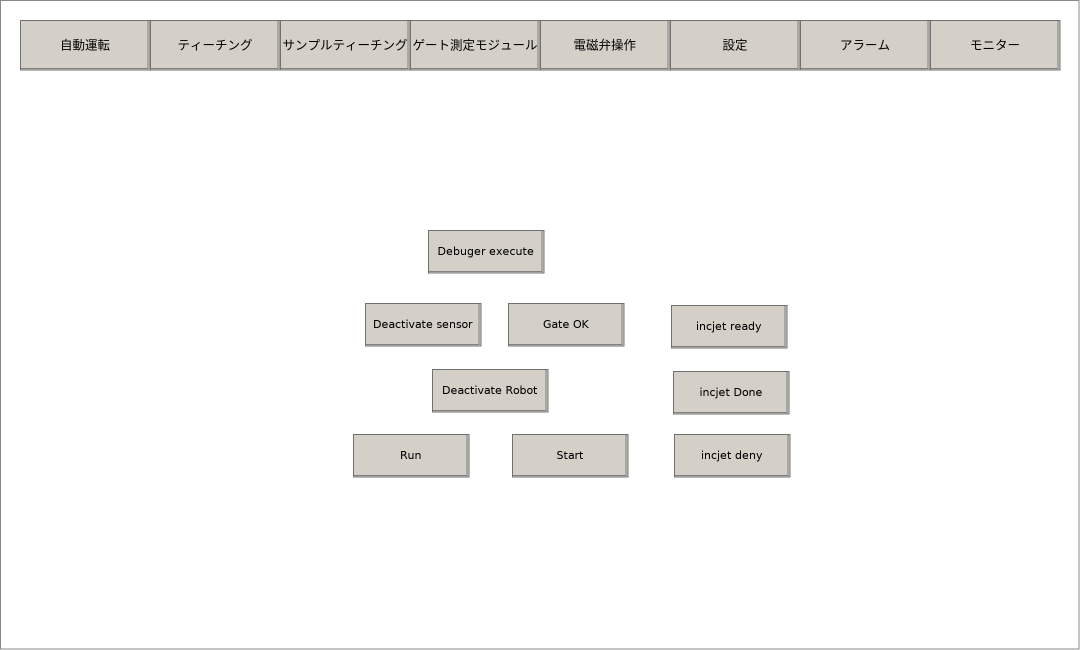
VISUALIZATION s_debug  // 1080x650
    Rectangle (0,0 1080x650)
    Button (20,20 130x50), "自動運転"
        OnMouseClick: change screen: s_auto
    Button (150,20 130x50), "ティーチング"
        OnMouseClick: change screen: s_teaching1
    Button (670,20 130x50), "設定"
        OnMouseClick: change screen: s_setting
    Button (540,20 130x50), "電磁弁操作"
        OnMouseClick: change screen: s_manual
    Button (410,20 130x50), "ゲート測定モジュール"
        OnMouseClick: change screen: s_gm_teaching
    Button (800,20 130x50), "アラーム", colour toggle: gvl_io.flg_signalTowerRed
        OnMouseClick: change screen: s_alarm
    Button (280,20 130x50), "サンプルティーチング"
        OnMouseClick: change screen: s_sample
    Button (930,20 130x50), "モニター"
        OnMouseClick: change screen: s_monitor
    Button (365,303 116x43), "Deactivate sensor", colour toggle: gvl_visu.flg_btn_vacSensOn
        toggle gvl_visu.flg_btn_vacSensOn
    Button (428,230 116x43), "Debuger execute", colour toggle: gvl_debug.flg_debug_run
        toggle gvl_debug.flg_debug_run
    Button (353,434 116x43), "Run", colour toggle: gvl_debug.flg_debug_start
        toggle gvl_debug.flg_debug_start
    Button (508,303 116x43), "Gate OK", colour toggle: gvl_debug.gateLengthISSuccessed
        toggle gvl_debug.gateLengthISSuccessed
    Button (512,434 116x43), "Start", colour toggle: gvl_debug.lensSetDone
        toggle gvl_debug.lensSetDone
    Button (671,305 116x43), "incjet ready", colour toggle: gvl_debug.flg_stampReady
        toggle gvl_debug.flg_stampReady
    Button (673,371 116x43), "incjet Done", colour toggle: gvl_debug.flg_stampDone
        tap gvl_debug.flg_stampDone
    Button (674,434 116x43), "incjet deny", colour toggle: gvl_gm.var_incjetInfo.flg_denyStamp
        toggle gvl_gm.var_incjetInfo.flg_denyStamp
    Button (432,369 116x43), "Deactivate Robot", colour toggle: gvl_visu.flg_btn_vacRobotOn
        toggle gvl_visu.flg_btn_vacRobotOn
END_VISUALIZATION

(* stored: Version 1.1.0.1, ProductVersion 3.1.4024.11
   Visu s_debug: Id {2b5719fb-3381-4cc2-825c-9b55c0761363} *)
